(* IEC 61131-3 sources: AXOpen/src/components.ur.robotics/ctrl/src/AxoUrCb3/v_3_x_x (part 2) *)

            Inputs.Zone                                             := Inputs.Inputs.Ints.Register_0;
            Inputs.InPosition                                       := Inputs.Inputs.Ints.Register_1;

           //Movement parameters
            Inputs.ActionNo                                         := Inputs.Inputs.Ints.Register_2;
            Inputs.GlobalSpeed                                      := Inputs.Inputs.Ints.Register_3;
            Inputs.ToolNo                                           := Inputs.Inputs.Ints.Register_4;
            Inputs.WorkobjectNo                                     := Inputs.Inputs.Ints.Register_5;
            Inputs.PointNo                                          := Inputs.Inputs.Ints.Register_6;

            Inputs.UserSpecSpeed1                                   := Inputs.Inputs.Floats.Register_0;
            Inputs.UserSpecSpeed2                                   := Inputs.Inputs.Floats.Register_1;
            Inputs.Coordinates.X                                    := Inputs.Inputs.Floats.Register_2;
            Inputs.Coordinates.Y                                    := Inputs.Inputs.Floats.Register_3;
            Inputs.Coordinates.Z                                    := Inputs.Inputs.Floats.Register_4;
            Inputs.Coordinates.Rx                                   := Inputs.Inputs.Floats.Register_5;
            Inputs.Coordinates.Ry                                   := Inputs.Inputs.Floats.Register_6;
            Inputs.Coordinates.Rz                                   := Inputs.Inputs.Floats.Register_7;

            //*************StartAtMainTask***************
            StartAtMainTask.SetIsDisabled(_stopTasksAreActive);
            IF StartAtMainTask.StartTriggered() THEN
                Status.Action.Id :=  UINT#100;
            END_IF;
            Messenger.ActivateOnCondition(ULINT#100,StartAtMainTask.IsBusy(), eAxoMessageCategory#Info);
            Messenger.ActivateOnCondition(ULINT#101,StartAtMainTask.IsDone(), eAxoMessageCategory#Info);
            IF StartAtMainTask.Execute(THIS) THEN
                _blink.Blink(Context := _context, inOnTime:=T#500MS,inOffTime:=T#500MS);
                IF _power_progress = 0 THEN
                    Status.Error.Id := UINT#0;
                    TaskMessenger.Restore();
                    THIS.CallTimers(FALSE);
                    _power_progress := 300;
                END_IF;
                // Start at main running: waiting for 'NORMAL' or 'REDUCED' mode is choosen.
                IF _power_progress = 300 THEN
                    IF _infoTimer.output THEN
                        IF NOT Inputs.Inputs.Safety.NO_IsNormalMode THEN
                            TaskMessenger.Activate( UINT#500, eAxoMessageCategory#Potential);
                            Status.Error.Id :=      UINT#500;
                        END_IF;
                        IF NOT Inputs.Inputs.Safety.RD_IsReducedMode THEN
                            TaskMessenger.Activate( UINT#501, eAxoMessageCategory#Potential);
                            Status.Error.Id :=      UINT#501;
                        END_IF;
                    END_IF;

                    IF Inputs.Inputs.Safety.NO_IsNormalMode OR Inputs.Inputs.Safety.RD_IsReducedMode THEN
                        THIS.CallTimers(FALSE);
                        _power_progress:=302;
                    END_IF;
                END_IF;
                // Start at main running: waiting for the program to start running.
                IF _power_progress = 302 THEN
                    IF _infoTimer.output THEN
                        TaskMessenger.Activate( UINT#502, eAxoMessageCategory#Potential);
                        Status.Error.Id :=      UINT#502;
                    END_IF;

                    Outputs.Start:=_blink.output;

                    IF Inputs.Inputs.Robot.PR_IsProgramRunning THEN
                        Outputs.Start := FALSE;
                        THIS.CallTimers(FALSE);
                        _power_progress:=303;
                    END_IF;
                END_IF;
                // Start at main finished.
                IF _power_progress = 303 THEN
                    StartAtMainTask.DoneWhen(TRUE);
                    THIS.CallTimers(FALSE);
                    _power_progress := 0;
                END_IF;

                THIS.CallTimers(TRUE);
                StartAtMainTask.ThrowWhen(_errorTimer.output );
                Status.Action.Id := TO_UINT(_power_progress);
                StartAtMainTask.ThrowWhen(StartAtMainTask.Duration >= Config.TaskTimeout AND Config.TaskTimeout > T#0s ,'<#StartAtMainTask timeout.#>');
            END_IF;
            IF StartAtMainTask.DoneReached() THEN
                Status.Action.Id :=  UINT#101;
                Status.Error.Id :=  UINT#0;
            ELSIF StartAtMainTask.ErrorOccured() THEN
                Status.Action.Id :=  UINT#10000;
                Status.Error.Id  :=  UINT#10000;
            ELSIF StartAtMainTask.AbortTriggered()THEN
                Status.Action.Id :=  UINT#10001;
                Status.Error.Id  :=  UINT#10001;
            END_IF;
            Messenger.ActivateOnCondition(ULINT#10000,StartAtMainTask.HasError(), eAxoMessageCategory#Error);
            Messenger.ActivateOnCondition(ULINT#10001,StartAtMainTask.IsAborted(), eAxoMessageCategory#Info);
            Messenger.ActivateOnCondition(ULINT#102,StartAtMainTask.RestoreTriggered() , eAxoMessageCategory#Info);
            IF StartAtMainTask.RestoreTriggered() AND _power_progress >= 300 AND _power_progress <= 309  THEN
                Status.Action.Id :=  UINT#102;
                _power_progress := 0;
            END_IF;
            //*******************************************

            //***********StartMotorsAndProgramTask*******
            StartMotorsAndProgramTask.SetIsDisabled(_stopTasksAreActive);
            IF StartMotorsAndProgramTask.StartTriggered() THEN
                Status.Action.Id :=  UINT#110;
            END_IF;
            Messenger.ActivateOnCondition(ULINT#110,StartMotorsAndProgramTask.IsBusy(), eAxoMessageCategory#Info);
            Messenger.ActivateOnCondition(ULINT#111,StartMotorsAndProgramTask.IsDone(), eAxoMessageCategory#Info);
            IF StartMotorsAndProgramTask.Execute(THIS) THEN
                _blink.Blink(Context := _context, inOnTime:=T#500MS,inOffTime:=T#500MS);

                IF _power_progress = 0 THEN
                    Status.Error.Id := UINT#0;
                    TaskMessenger.Restore();
                    THIS.CallTimers(FALSE);
                    _power_progress := 310;
                END_IF;
                // Start motors and program running: waiting for 'NORMAL' or 'REDUCED' mode is choosen.
                IF _power_progress = 310 THEN
                    IF _infoTimer.output THEN
                        IF NOT Inputs.Inputs.Safety.NO_IsNormalMode THEN
                            TaskMessenger.Activate( UINT#510, eAxoMessageCategory#Potential);
                            Status.Error.Id :=      UINT#510;
                        END_IF;
                        IF NOT Inputs.Inputs.Safety.RD_IsReducedMode THEN
                            TaskMessenger.Activate( UINT#511, eAxoMessageCategory#Potential);
                            Status.Error.Id :=      UINT#511;
                        END_IF;
                    END_IF;

                    IF Inputs.Inputs.Safety.NO_IsNormalMode OR Inputs.Inputs.Safety.RD_IsReducedMode THEN
                        THIS.CallTimers(FALSE);
                        _power_progress:=312;
                    END_IF;
                END_IF;
                // Start motors and program running: waiting for the error to be reset (on the robot teach pendant).
                IF _power_progress = 312 THEN
                    IF _infoTimer.output THEN
                        TaskMessenger.Activate( UINT#512, eAxoMessageCategory#Potential);
                        Status.Error.Id :=      UINT#512;
                    END_IF;

                    IF NOT Inputs.Inputs.Safety.FT_IsFault THEN
                        THIS.CallTimers(FALSE);
                        _power_progress := 313;
                    END_IF;
                END_IF;
                // Start motors and program running: waiting for the emergency stop error to be reset (on the robot teach pendant).
                IF _power_progress = 313 THEN
                    IF _infoTimer.output THEN
                        IF Inputs.Inputs.Safety.ES_IsEmergencyStopped  THEN
                            TaskMessenger.Activate( UINT#513, eAxoMessageCategory#Potential);
                            Status.Error.Id :=      UINT#513;
                        END_IF;
                        IF Inputs.Inputs.Safety.PS_IsProtectiveStopped  THEN
                            TaskMessenger.Activate( UINT#514, eAxoMessageCategory#Potential);
                            Status.Error.Id :=      UINT#514;
                        END_IF;
                        IF Inputs.Inputs.Safety.SS_IsSafeguardStopped  THEN
                            TaskMessenger.Activate( UINT#515, eAxoMessageCategory#Potential);
                            Status.Error.Id :=      UINT#515;
                        END_IF;
                        IF Inputs.Inputs.Safety.RC_IsRecoveryMode  THEN
                            TaskMessenger.Activate( UINT#516, eAxoMessageCategory#Potential);
                            Status.Error.Id :=      UINT#516;
                        END_IF;
                        IF Inputs.Inputs.Safety.ST_IsStoppedDueSafety  THEN
                            TaskMessenger.Activate( UINT#517, eAxoMessageCategory#Potential);
                            Status.Error.Id :=      UINT#517;
                        END_IF;
                        IF Inputs.Inputs.Safety.VL_IsViolation  THEN
                            TaskMessenger.Activate( UINT#518, eAxoMessageCategory#Potential);
                            Status.Error.Id :=      UINT#518;
                        END_IF;
                    END_IF;

                    IF NOT Inputs.Inputs.Safety.ES_IsEmergencyStopped
                        AND NOT Inputs.Inputs.Safety.PS_IsProtectiveStopped
                        AND NOT Inputs.Inputs.Safety.SS_IsSafeguardStopped
                        AND NOT Inputs.Inputs.Safety.RC_IsRecoveryMode
                        AND NOT Inputs.Inputs.Safety.ST_IsStoppedDueSafety
                        AND NOT Inputs.Inputs.Safety.VL_IsViolation THEN
                        THIS.CallTimers(FALSE);
                        _power_progress := 319;
                    END_IF;
                END_IF;
                // Start motors and program running: waiting for the motors to be powered on.
                IF _power_progress = 319 THEN
                    IF _infoTimer.output THEN
                        TaskMessenger.Activate( UINT#519, eAxoMessageCategory#Potential);
                        Status.Error.Id :=      UINT#519;
                    END_IF;

                    Outputs.MotorOn:=_blink.output;

                    IF Inputs.Inputs.Safety.FT_IsFault THEN
                        THIS.CallTimers(FALSE);
                        _power_progress := 310;
                    END_IF;

                    IF Inputs.Inputs.Robot.PW_IsPowerOn THEN
                         Outputs.MotorOn:=FALSE;
                         THIS.CallTimers(FALSE);
                         _power_progress := 320;
                    END_IF;
                END_IF;
                // Start motors and program running: waiting for the motors to be powered on.
                IF _power_progress = 320 THEN
                    IF _infoTimer.output THEN
                        TaskMessenger.Activate( UINT#520, eAxoMessageCategory#Potential);
                        Status.Error.Id :=      UINT#520;
                    END_IF;

                    Outputs.MotorOn:=_blink.output;

                    IF Inputs.Inputs.Safety.FT_IsFault THEN
                        THIS.CallTimers(FALSE);
                        _power_progress := 310;
                    END_IF;

                    IF Inputs.Inputs.Robot.PW_IsPowerOn THEN
                         Outputs.MotorOn:=FALSE;
                         THIS.CallTimers(FALSE);
                         _power_progress := 321;
                    END_IF;
                END_IF;
                // Start motors and program running: waiting for the program to start running.
                IF _power_progress = 321 THEN
                    IF _infoTimer.output THEN
                        TaskMessenger.Activate( UINT#521, eAxoMessageCategory#Potential);
                        Status.Error.Id :=      UINT#521;
                    END_IF;

                    Outputs.Start:=_blink.output;

                    IF Inputs.Inputs.Safety.FT_IsFault THEN
                        THIS.CallTimers(FALSE);
                        _power_progress := 310;
                    END_IF;

                    IF Inputs.Inputs.Robot.PR_IsProgramRunning AND NOT Inputs.Inputs.Safety.FT_IsFault THEN
                         Outputs.Start:=FALSE;
                         THIS.CallTimers(FALSE);
                         _power_progress := 322;
                    END_IF;
                END_IF;
                // Start motors and program finished.
                IF _power_progress = 322 THEN
                    StartMotorsAndProgramTask.DoneWhen(TRUE);
                    THIS.CallTimers(FALSE);
                    _power_progress := 0;
                END_IF;

                THIS.CallTimers(TRUE);
                StartMotorsAndProgramTask.ThrowWhen(_errorTimer.output);
                Status.Action.Id := TO_UINT(_power_progress);
                StartMotorsAndProgramTask.ThrowWhen(StartMotorsAndProgramTask.Duration >= Config.TaskTimeout AND Config.TaskTimeout > T#0s ,'<#StartMotorsAndProgramTask timeout.#>');
            END_IF;
            IF StartMotorsAndProgramTask.DoneReached() THEN
                Status.Action.Id :=  UINT#111;
                Status.Error.Id :=  UINT#0;
            ELSIF StartMotorsAndProgramTask.ErrorOccured() THEN
                Status.Action.Id :=  UINT#10010;
                Status.Error.Id  :=  UINT#10010;
            ELSIF StartMotorsAndProgramTask.AbortTriggered() THEN
                Status.Action.Id :=  UINT#10011;
                Status.Error.Id  :=  UINT#10011;
            END_IF;
            Messenger.ActivateOnCondition(ULINT#10010,StartMotorsAndProgramTask.HasError(), eAxoMessageCategory#Error);
            Messenger.ActivateOnCondition(ULINT#10011,StartMotorsAndProgramTask.IsAborted(), eAxoMessageCategory#Info);
            Messenger.ActivateOnCondition(ULINT#112,StartMotorsAndProgramTask.RestoreTriggered() , eAxoMessageCategory#Info);
            IF StartMotorsAndProgramTask.RestoreTriggered() AND _power_progress >= 310 AND _power_progress <= 329  THEN
                Status.Action.Id :=  UINT#112;
                _power_progress := 0;
            END_IF;
            //*******************************************

            //***********StartMovementsTask**************
            StartMovementsTask.SetIsDisabled(NOT Inputs.Inputs.Robot.PW_IsPowerOn);
            IF StartMovementsTask.StartTriggered() THEN
                Status.Action.Id :=  UINT#180;
            END_IF;
            Messenger.ActivateOnCondition(ULINT#180,StartMovementsTask.IsBusy(), eAxoMessageCategory#Info);
            Messenger.ActivateOnCondition(ULINT#181,StartMovementsTask.IsDone(), eAxoMessageCategory#Info);
            IF StartMovementsTask.Execute(THIS) THEN
                IF _movement_progress = 0 THEN
                    Status.Error.Id :=  UINT#0;
                    TaskMessenger.Restore();
                    THIS.CallTimers(FALSE);
                    _movement_progress := 380;
                END_IF;
                // Start movements running: waiting for the program to start running.
                IF _movement_progress = 380 THEN
                    IF _infoTimer.output THEN
                        TaskMessenger.Activate( UINT#580, eAxoMessageCategory#Potential);
                        Status.Error.Id :=      UINT#580;
                    END_IF;

                    IF Inputs.Inputs.Robot.PR_IsProgramRunning THEN
                        THIS.CallTimers(FALSE);
                        _movement_progress := 381;
                    END_IF;
                END_IF;
                // Start movements running: waiting for the motors to be powered on.
                IF _movement_progress = 381 THEN
                    IF _infoTimer.output THEN
                        TaskMessenger.Activate( UINT#581, eAxoMessageCategory#Potential);
                        Status.Error.Id :=      UINT#581;
                    END_IF;

                    IF Inputs.Inputs.Robot.PW_IsPowerOn THEN
                        THIS.CallTimers(FALSE);
                        _movement_progress := 382;
                    END_IF;
                END_IF;
                // Start movements running: waiting for the error to be reset (on the robot teach pendant).
                IF _movement_progress = 382 THEN
                    IF _infoTimer.output THEN
                        TaskMessenger.Activate( UINT#582, eAxoMessageCategory#Potential);
                        Status.Error.Id :=      UINT#582;
                    END_IF;

                    IF NOT Inputs.Inputs.Safety.FT_IsFault THEN
                        THIS.CallTimers(FALSE);
                        _movement_progress := 383;
                    END_IF;
                END_IF;
                // Start movements running: sending parameters of the movement to the controller.
                IF _movement_progress = 383 THEN
                    IF _infoTimer.output THEN
                        TaskMessenger.Activate( UINT#583, eAxoMessageCategory#Potential);
                        Status.Error.Id :=      UINT#583;
                    END_IF;

                    Outputs.GlobalSpeed     := TO_DINT(Status.CurrentMovementParameters.GlobalSpeed);
                    Outputs.ToolNo          := TO_DINT(Status.CurrentMovementParameters.ToolNo);
                    Outputs.WorkobjectNo    := TO_DINT(Status.CurrentMovementParameters.WorkobjectNo);
                    Outputs.PointNo         := TO_DINT(Status.CurrentMovementParameters.PointNo);
                    Outputs.UserSpecSpeed1  := Status.CurrentMovementParameters.UserSpecSpeed1;
                    Outputs.UserSpecSpeed2  := Status.CurrentMovementParameters.UserSpecSpeed2;
                    Outputs.Coordinates     := Status.CurrentMovementParameters.Coordinates;

                    Outputs.ActionNo := DINT#254;

                    IF Outputs.ActionNo = Inputs.ActionNo THEN
                        THIS.CallTimers(FALSE);
                        _movement_progress := 384;
                    END_IF;
                END_IF;
                // Start movements running: waiting for the movement parameters sent to the controller to be mirrored back.
                IF _movement_progress = 384 THEN
                    IF _infoTimer.output THEN
                        IF Inputs.GlobalSpeed <> TO_DINT(Status.CurrentMovementParameters.GlobalSpeed) THEN
                            TaskMessenger.Activate( UINT#584, eAxoMessageCategory#Potential);
                            Status.Error.Id :=      UINT#584;//<#Waiting for Inputs.GlobalSpeed to be equal to MovementParameters.GlobalSpeed!
                        END_IF;
                        IF Inputs.ToolNo <> TO_DINT(Status.CurrentMovementParameters.ToolNo) THEN
                            TaskMessenger.Activate( UINT#585, eAxoMessageCategory#Potential);
                            Status.Error.Id :=      UINT#585;//<#Waiting for Inputs.ToolNo to be equal to MovementParameters.ToolNo!
                        END_IF;
                        IF Inputs.WorkobjectNo <> TO_DINT(Status.CurrentMovementParameters.WorkobjectNo) THEN
                            TaskMessenger.Activate( UINT#586, eAxoMessageCategory#Potential);
                            Status.Error.Id :=      UINT#586;//<#Waiting for Inputs.WorkobjectNo to be equal to MovementParameters.WorkobjectNo!
                        END_IF;
                        IF Inputs.PointNo <> TO_DINT(Status.CurrentMovementParameters.PointNo) THEN
                            TaskMessenger.Activate( UINT#587, eAxoMessageCategory#Potential);
                            Status.Error.Id :=      UINT#587;//<#Waiting for Inputs.PointNo to be equal to MovementParameters.PointNo!
                        END_IF;
                        IF Inputs.UserSpecSpeed1 <> Status.CurrentMovementParameters.UserSpecSpeed1 THEN
                            TaskMessenger.Activate( UINT#588, eAxoMessageCategory#Potential);
                            Status.Error.Id :=      UINT#588;//<#Waiting for Inputs.UserSpecSpeed1 to be equal to MovementParameters.UserSpecSpeed1!
                        END_IF;
                        IF Inputs.UserSpecSpeed2 <> Status.CurrentMovementParameters.UserSpecSpeed2 THEN
                            TaskMessenger.Activate( UINT#589, eAxoMessageCategory#Potential);
                            Status.Error.Id :=      UINT#589;//<#Waiting for Inputs.UserSpecSpeed2 to be equal to MovementParameters.UserSpecSpeed2!
                        END_IF;
                    END_IF;

                    IF 	Inputs.GlobalSpeed      = TO_DINT(Status.CurrentMovementParameters.GlobalSpeed) AND
                        Inputs.ToolNo           = TO_DINT(Status.CurrentMovementParameters.ToolNo) AND
                        Inputs.WorkobjectNo     = TO_DINT(Status.CurrentMovementParameters.WorkobjectNo) AND
                        Inputs.PointNo          = TO_DINT(Status.CurrentMovementParameters.PointNo) AND
                        Inputs.UserSpecSpeed1   = Status.CurrentMovementParameters.UserSpecSpeed1 AND
                        Inputs.UserSpecSpeed2   = Status.CurrentMovementParameters.UserSpecSpeed2 AND
                        AXOpen.Components.Robotics.CoordinatesAreNearlyEqual(Inputs.Coordinates,Status.CurrentMovementParameters.Coordinates,REAL#0.01,REAL#0.01,REAL#0.01,REAL#0.01,REAL#0.01,REAL#0.01) THEN
                        THIS.CallTimers(FALSE);
                        _movement_progress:=390;
                    END_IF;
                END_IF;
                // Start movements running: acknowleadging of the movement parameters.
                IF _movement_progress = 390 THEN
                    IF _infoTimer.output THEN
                        TaskMessenger.Activate( UINT#590, eAxoMessageCategory#Potential);
                        Status.Error.Id :=      UINT#590;
                    END_IF;

                    Outputs.ActionNo := DINT#255;

                    IF Outputs.ActionNo = Inputs.ActionNo THEN
                        THIS.CallTimers(FALSE);
                        _movement_progress:=391;
                    END_IF;
                END_IF;
                // Start movements running: waiting for the movement is finished.
                IF _movement_progress = 391 THEN
                    IF _infoTimer.output THEN
                        TaskMessenger.Activate( UINT#591, eAxoMessageCategory#Potential);
                        Status.Error.Id :=      UINT#591;
                    END_IF;

                    Outputs.ActionNo := TO_DINT(Status.CurrentMovementParameters.ActionNo);

                    IF Outputs.ActionNo = Inputs.ActionNo THEN
                        THIS.CallTimers(FALSE);
                        _movement_progress:=392;
                    END_IF;
                END_IF;
                // Start movements running: acknowleadging of the finished movement.
                IF _movement_progress = 392 THEN
                    IF _infoTimer.output THEN
                        TaskMessenger.Activate( UINT#592, eAxoMessageCategory#Potential);
                        Status.Error.Id :=      UINT#592;
                    END_IF;

                    Outputs.ActionNo := DINT#255;

                    IF Outputs.ActionNo = Inputs.ActionNo THEN
                        _movement_progress := 0;
                        StartMovementsTask.DoneWhen(TRUE);
                    END_IF;
                END_IF;

	            THIS.CallTimers(TRUE);

                StartMovementsTask.ThrowWhen(_errorTimer.output);
                Status.Action.Id := TO_UINT(_movement_progress);
                StartMovementsTask.ThrowWhen(StartMovementsTask.Duration >= Config.TaskTimeout AND Config.TaskTimeout > T#0s ,'<#StartMovementsTask timeout.#>');
            END_IF;
            IF StartMovementsTask.DoneReached() THEN
                Status.Action.Id :=  UINT#181;
                Status.Error.Id :=  UINT#0;
            ELSIF StartMovementsTask.ErrorOccured() THEN
                Status.Action.Id :=  UINT#10080;
                Status.Error.Id  :=  UINT#10080;
            ELSIF StartMovementsTask.AbortTriggered()THEN
                Status.Action.Id :=  UINT#10081;
                Status.Error.Id  :=  UINT#10081;
            END_IF;
            Messenger.ActivateOnCondition(ULINT#10080,StartMovementsTask.HasError(), eAxoMessageCategory#Error);
            Messenger.ActivateOnCondition(ULINT#10081,StartMovementsTask.IsAborted(), eAxoMessageCategory#Info);
            Messenger.ActivateOnCondition(ULINT#182,StartMovementsTask.RestoreTriggered() , eAxoMessageCategory#Info);
            IF StartMovementsTask.RestoreTriggered() AND _movement_progress >= 380 AND _movement_progress <= 399  THEN
                Status.Action.Id :=  UINT#182;
                _movement_progress := 0;
            END_IF;
            //*******************************************

            //***********StopMovementsAndProgramTask*****
            StopMovementsAndProgramTask.SetIsDisabled(FALSE);
            IF StopMovementsAndProgramTask.StartTriggered() THEN
                Status.Action.Id :=  UINT#210;
            END_IF;
            Messenger.ActivateOnCondition(ULINT#210,StopMovementsAndProgramTask.IsBusy(), eAxoMessageCategory#Info);
            Messenger.ActivateOnCondition(ULINT#211,StopMovementsAndProgramTask.IsDone(), eAxoMessageCategory#Info);
            IF StopMovementsAndProgramTask.Execute(THIS) THEN
                IF _power_progress = 0 THEN
                    Status.Error.Id :=  UINT#0;
                    TaskMessenger.Restore();
                    THIS.CallTimers(FALSE);
                    _power_progress := 410;
                END_IF;
                // Stop movements and program running: waiting for 'NORMAL' or 'REDUCED' mode is choosen.
                IF _power_progress = 410 THEN
                    IF _infoTimer.output THEN
                        IF NOT Inputs.Inputs.Safety.NO_IsNormalMode THEN
                            TaskMessenger.Activate( UINT#610, eAxoMessageCategory#Potential);
                            Status.Error.Id :=      UINT#610;
                        END_IF;
                        IF NOT Inputs.Inputs.Safety.RD_IsReducedMode THEN
                            TaskMessenger.Activate( UINT#611, eAxoMessageCategory#Potential);
                            Status.Error.Id :=      UINT#611;
                        END_IF;
                    END_IF;

                    IF Inputs.Inputs.Safety.NO_IsNormalMode OR Inputs.Inputs.Safety.RD_IsReducedMode THEN
                        THIS.CallTimers(FALSE);
                        _power_progress:=412;
                    END_IF;
                END_IF;
                // Stop movements and program running: waiting for the program to be stopped."
                IF _power_progress = 412 THEN
                    IF _infoTimer.output THEN
                        TaskMessenger.Activate( UINT#612, eAxoMessageCategory#Potential);
                        Status.Error.Id :=      UINT#612;
                    END_IF;

                    Outputs.Stop := TRUE;

                    IF NOT Inputs.Inputs.Robot.PR_IsProgramRunning THEN
                        Outputs.Stop := FALSE ;
                        THIS.CallTimers(FALSE);
                        _power_progress:=413;
                    END_IF;
                END_IF;
                // Stop movements and program finished.
                IF _power_progress = 413 THEN
                    Outputs.Stop := FALSE ;
                    StopMovementsAndProgramTask.DoneWhen(TRUE);
                    _power_progress := 0;
                END_IF;

                THIS.CallTimers(TRUE);
                StopMovementsAndProgramTask.ThrowWhen(_errorTimer.output);
                Status.Action.Id := TO_UINT(_power_progress);
                StopMovementsAndProgramTask.ThrowWhen(StopMovementsAndProgramTask.Duration >= Config.TaskTimeout AND Config.TaskTimeout > T#0s ,'<#StopMovementsAndProgramTask timeout.#>');
            END_IF;
            IF StopMovementsAndProgramTask.DoneReached() THEN
                Status.Action.Id :=  UINT#211;
                Status.Error.Id :=  UINT#0;
            ELSIF StopMovementsAndProgramTask.ErrorOccured() THEN
                Status.Action.Id :=  UINT#10110;
                Status.Error.Id  :=  UINT#10110;
            ELSIF StopMovementsAndProgramTask.AbortTriggered()THEN
                Status.Action.Id :=  UINT#10111;
                Status.Error.Id  :=  UINT#10111;
            END_IF;
            Messenger.ActivateOnCondition(ULINT#10110,StopMovementsAndProgramTask.HasError(), eAxoMessageCategory#Error);
            Messenger.ActivateOnCondition(ULINT#10111,StopMovementsAndProgramTask.IsAborted(), eAxoMessageCategory#Info);
            Messenger.ActivateOnCondition(ULINT#212,StopMovementsAndProgramTask.RestoreTriggered() , eAxoMessageCategory#Info);
            IF StopMovementsAndProgramTask.RestoreTriggered() AND _power_progress >= 410 AND _power_progress <= 419  THEN
                Status.Action.Id :=  UINT#212;
                _power_progress := 0;
            END_IF;
            //*******************************************

            //***********StopMovementsTask***************
            StopMovementsTask.SetIsDisabled(FALSE);
            IF StopMovementsAndProgramTask.StartTriggered() THEN
                Status.Action.Id :=  UINT#220;
            END_IF;
            Messenger.ActivateOnCondition(ULINT#220,StopMovementsAndProgramTask.IsBusy(), eAxoMessageCategory#Info);
            Messenger.ActivateOnCondition(ULINT#221,StopMovementsAndProgramTask.IsDone(), eAxoMessageCategory#Info);
            IF StopMovementsTask.Execute(THIS) THEN
                IF _power_progress = 0 THEN
                    Status.Error.Id :=  UINT#0;
                    TaskMessenger.Restore();
                    THIS.CallTimers(FALSE);
                    _power_progress := 420;
                END_IF;
                // Stop movements running: waiting for 'NORMAL' or 'REDUCED' mode is choosen.
                IF _power_progress = 420 THEN
                    IF _infoTimer.output THEN
                        IF NOT Inputs.Inputs.Safety.NO_IsNormalMode THEN
                            TaskMessenger.Activate( UINT#620, eAxoMessageCategory#Potential);
                            Status.Error.Id :=      UINT#620;
                        END_IF;
                        IF NOT Inputs.Inputs.Safety.RD_IsReducedMode THEN
                            TaskMessenger.Activate( UINT#621, eAxoMessageCategory#Potential);
                            Status.Error.Id :=      UINT#621;
                        END_IF;
                    END_IF;

                    IF Inputs.Inputs.Safety.NO_IsNormalMode OR Inputs.Inputs.Safety.RD_IsReducedMode THEN
                        THIS.CallTimers(FALSE);
                        _power_progress:=422;
                    END_IF;
                END_IF;
                // Stop movements running: waiting for the program to be stopped.
                IF _power_progress = 422 THEN
                    IF _infoTimer.output THEN
                        TaskMessenger.Activate( UINT#622, eAxoMessageCategory#Potential);
                        Status.Error.Id :=      UINT#622;
                    END_IF;

                    Outputs.Pause := TRUE;

                    IF NOT Inputs.Inputs.Robot.PR_IsProgramRunning THEN
                        Outputs.Pause := FALSE ;
                        THIS.CallTimers(FALSE);
                        _power_progress:=423;
                    END_IF;
                END_IF;
                // Stop movements finished.
                IF _power_progress = 423 THEN
                    Outputs.Pause := FALSE ;
                    StopMovementsTask.DoneWhen(TRUE);
                    _power_progress := 0;
                END_IF;

                THIS.CallTimers(TRUE);
                StopMovementsTask.ThrowWhen(_errorTimer.output);
                Status.Action.Id := TO_UINT(_power_progress);
                StopMovementsTask.ThrowWhen(StopMovementsTask.Duration >= Config.TaskTimeout AND Config.TaskTimeout > T#0s ,'<#StopMovementsTask timeout.#>');
            END_IF;
            IF StopMovementsTask.DoneReached() THEN
                Status.Action.Id :=  UINT#221;
                Status.Error.Id :=  UINT#0;
            ELSIF StopMovementsTask.ErrorOccured() THEN
                Status.Action.Id :=  UINT#10120;
                Status.Error.Id  :=  UINT#10120;
            ELSIF StopMovementsTask.AbortTriggered()THEN
                Status.Action.Id :=  UINT#10121;
                Status.Error.Id  :=  UINT#10121;
            END_IF;
            Messenger.ActivateOnCondition(ULINT#10120,StopMovementsTask.HasError(), eAxoMessageCategory#Error);
            Messenger.ActivateOnCondition(ULINT#10121,StopMovementsTask.IsAborted(), eAxoMessageCategory#Info);
            Messenger.ActivateOnCondition(ULINT#222,StopMovementsTask.RestoreTriggered() , eAxoMessageCategory#Info);
            IF StopMovementsTask.RestoreTriggered() AND _power_progress >= 420 AND _power_progress <= 429  THEN
                Status.Action.Id :=  UINT#222;
                _power_progress := 0;
            END_IF;
            //*******************************************

            //*************POWER ON********************
            PowerOnTask.SetIsDisabled(NOT(Inputs.RobotMode=eAxoUrRoboticsRobotMode#DISCONNECTED AND Config.RemotePowerOnEnabled));
            IF PowerOnTask.Execute(THIS) THEN
                refPowerOnPulse^ :=TRUE;
                Status.Action.Id :=  UINT#420;//('<#POWER ON PULSE WAS SEND TO CONTROLER#>');
                PowerOnTask.DoneWhen(PowerOnTask.Duration > Config.RemotePowerOnPulse);
            END_IF;

            IF refPowerOnPulse^ AND PowerOnTask.IsDone()  OR NOT Config.RemotePowerOnEnabled THEN
                refPowerOnPulse^ :=FALSE;
            END_IF;

            //****************************************

            _someTaskIsActive := StartAtMainTask.IsBusy()
                                OR StartMotorsAndProgramTask.IsBusy()
                                OR StartMovementsTask.IsBusy()
                                OR StopMovementsTask.IsBusy()
                                OR StopMovementsAndProgramTask.IsBusy();

            IF _someTaskIsActive THEN
                IF(Inputs.Inputs.Safety.ES_IsEmergencyStopped) THEN
                    Messenger.Activate(UINT#2000, eAxoMessageCategory#Error);
                    Status.Error.Id := UINT#2000;
                END_IF;
                IF(Inputs.Inputs.Safety.ST_IsStoppedDueSafety) THEN
                    Messenger.Activate(UINT#2001, eAxoMessageCategory#Error);
                    Status.Error.Id := UINT#2001;
                END_IF;
            END_IF;
            //***********UPDATE**OUTPUTS*****************
            //SYSTEM OUTPUTS
            Outputs.Outputs.Reg1.Bit_0 := Outputs.Start;
            Outputs.outputs.Reg1.Bit_1 := Outputs.Stop;
            Outputs.outputs.Reg1.Bit_2 := Outputs.Pause;
            Outputs.outputs.Reg1.Bit_3 := Outputs.MotorOn;
            //Outputs.outputs.Reg1.Bit_4 := Outputs.RunAction;

            //Tool signals
            Outputs.Outputs.Reg1.Bit_8 := Outputs.Tool_1_Retract;
            Outputs.outputs.Reg1.Bit_9 := Outputs.Tool_1_Extend;
            Outputs.outputs.Reg1.Bit_10 := Outputs.Tool_2_Retract;
            Outputs.outputs.Reg1.Bit_11 := Outputs.Tool_2_Extend;
            Outputs.outputs.Reg1.Bit_12 := Outputs.Tool_3_Retract;
            Outputs.outputs.Reg1.Bit_13 := Outputs.Tool_3_Extend;
            Outputs.outputs.Reg1.Bit_14 := Outputs.Tool_4_Retract;
            Outputs.outputs.Reg1.Bit_15 := Outputs.Tool_4_Extend;

            //zone
            Outputs.Outputs.Reg1.Int_0 := Outputs.Zone;
            //position
            Outputs.Outputs.Reg1.Int_1 := Outputs.InPosition;

            //Movement parameters
            Outputs.Outputs.Reg1.Int_2 := Outputs.ActionNo;
            Outputs.Outputs.Reg1.Int_3 := Outputs.GlobalSpeed;
            Outputs.Outputs.Reg1.Int_4 := Outputs.ToolNo;
            Outputs.Outputs.Reg1.Int_5 := Outputs.WorkobjectNo;
            Outputs.Outputs.Reg1.Int_6 := Outputs.PointNo;
            //master mode  such as manual/auto ....
            Outputs.Outputs.Reg1.Int_7 := TO_DINT(Outputs.MasterMode);

            Outputs.Outputs.Reg1.Float_0 := Outputs.UserSpecSpeed1;
            Outputs.Outputs.Reg1.Float_1 := Outputs.UserSpecSpeed2;

            ////Coordinates
            Outputs.Outputs.Reg1.Float_2 := Outputs.Coordinates.X ;
            Outputs.Outputs.Reg1.Float_3 := Outputs.Coordinates.Y;
            Outputs.Outputs.Reg1.Float_4 := Outputs.Coordinates.Z ;
            Outputs.Outputs.Reg1.Float_5 := (Outputs.Coordinates.Rx);
            Outputs.Outputs.Reg1.Float_6 := (Outputs.Coordinates.Ry);
            Outputs.Outputs.Reg1.Float_7 := (Outputs.Coordinates.Rz);

            //st_URO_CB3_O2TSpeedData => 8_O2T Robot IO
            _data24[0].%X0 := Outputs.Outputs.Speed.SSM_SpeedSliderFractionMask;

            _dword := TO_DWORD(Outputs.Outputs.Speed.SpeedSliderFraction * REAL#0.01);
            _data24[4] := _dword.%B3;
            _data24[5] := _dword.%B2;
            _data24[6] := _dword.%B1;
            _data24[7] := _dword.%B0;

            //st_URO_CB3_O2TIoData => 8_O2T Robot IO
            _data24[8]  := TO_BYTE(Outputs.Outputs.IO.StandardDigitalOutputMask);
            _data24[9]  := TO_BYTE(Outputs.Outputs.IO.ConfigurableDigitalOutputMask);
            _data24[10] := TO_BYTE(Outputs.Outputs.IO.StandardDigitalOutputs);
            _data24[11] := TO_BYTE(Outputs.Outputs.IO.ConfigurableDdigitalOutputs);
            _data24[12] := TO_BYTE(Outputs.Outputs.IO.AOM_AnalogOutputMask);
            _data24[13] := TO_BYTE(Outputs.Outputs.IO.AOT_AnalogOutputTypes);
            _data24[14] := TO_BYTE(Outputs.Outputs.IO.TDOM_ToolDigitalOutputMask);
            _data24[15] := TO_BYTE(Outputs.Outputs.IO.TDO_ToolDigitalOutput);

            _dword := TO_DWORD(Outputs.Outputs.IO.StandardAnalogOutput_0);
            _data24[16] := _dword.%B3;
            _data24[17] := _dword.%B2;
            _data24[18] := _dword.%B1;
            _data24[19] := _dword.%B0;

            _dword := TO_DWORD(Outputs.Outputs.IO.StandardAnalogOutput_1);
            _data24[20] := _dword.%B3;
            _data24[21] := _dword.%B2;
            _data24[22] := _dword.%B1;
            _data24[23] := _dword.%B0;

            _retVal := Siemens.Simatic.DistributedIO.WriteData((Config.HWIDs.HwId_AxoUrRobotics_O2T_Robot_IO),_data24);
            IF _retVal > WORD#0 THEN
                Messenger.Activate(UINT#1231, eAxoMessageCategory#Error);
                Status.Error.Id := UINT#1231;
                RETURN;
            END_IF;

            //st_URO_CB3_O2TRegData => 9_O2T General Purpose Registers 1
            _data100[0].%X0 :=  Outputs.Outputs.Reg1.Bit_0;
            _data100[0].%X1 :=  Outputs.Outputs.Reg1.Bit_1;
            _data100[0].%X2 :=  Outputs.Outputs.Reg1.Bit_2;
            _data100[0].%X3 :=  Outputs.Outputs.Reg1.Bit_3;
            _data100[0].%X4 :=  Outputs.Outputs.Reg1.Bit_4;
            _data100[0].%X5 :=  Outputs.Outputs.Reg1.Bit_5;
            _data100[0].%X6 :=  Outputs.Outputs.Reg1.Bit_6;
            _data100[0].%X7 :=  Outputs.Outputs.Reg1.Bit_7;

            _data100[1].%X0 :=  Outputs.Outputs.Reg1.Bit_8;
            _data100[1].%X1 :=  Outputs.Outputs.Reg1.Bit_9;
            _data100[1].%X2 :=  Outputs.Outputs.Reg1.Bit_10;
            _data100[1].%X3 :=  Outputs.Outputs.Reg1.Bit_11;
            _data100[1].%X4 :=  Outputs.Outputs.Reg1.Bit_12;
            _data100[1].%X5 :=  Outputs.Outputs.Reg1.Bit_13;
            _data100[1].%X6 :=  Outputs.Outputs.Reg1.Bit_14;
            _data100[1].%X7 :=  Outputs.Outputs.Reg1.Bit_15;

            _data100[2].%X0 :=  Outputs.Outputs.Reg1.Bit_16;
            _data100[2].%X1 :=  Outputs.Outputs.Reg1.Bit_17;
            _data100[2].%X2 :=  Outputs.Outputs.Reg1.Bit_18;
            _data100[2].%X3 :=  Outputs.Outputs.Reg1.Bit_19;
            _data100[2].%X4 :=  Outputs.Outputs.Reg1.Bit_20;
            _data100[2].%X5 :=  Outputs.Outputs.Reg1.Bit_21;
            _data100[2].%X6 :=  Outputs.Outputs.Reg1.Bit_22;
            _data100[2].%X7 :=  Outputs.Outputs.Reg1.Bit_23;

            _data100[3].%X0 :=  Outputs.Outputs.Reg1.Bit_24;
            _data100[3].%X1 :=  Outputs.Outputs.Reg1.Bit_25;
            _data100[3].%X2 :=  Outputs.Outputs.Reg1.Bit_26;
            _data100[3].%X3 :=  Outputs.Outputs.Reg1.Bit_27;
            _data100[3].%X4 :=  Outputs.Outputs.Reg1.Bit_28;
            _data100[3].%X5 :=  Outputs.Outputs.Reg1.Bit_29;
            _data100[3].%X6 :=  Outputs.Outputs.Reg1.Bit_30;
            _data100[3].%X7 :=  Outputs.Outputs.Reg1.Bit_31;

            _dword          := TO_DWORD( Outputs.Outputs.Reg1.Int_0);
            _data100[4]     := _dword.%B3;
            _data100[5]     := _dword.%B2;
            _data100[6]     := _dword.%B1;
            _data100[7]     := _dword.%B0;

            _dword          := TO_DWORD( Outputs.Outputs.Reg1.Int_1);
            _data100[8]     := _dword.%B3;
            _data100[9]     := _dword.%B2;
            _data100[10]    := _dword.%B1;
            _data100[11]    := _dword.%B0;

            _dword          := TO_DWORD( Outputs.Outputs.Reg1.Int_2);
            _data100[12]    := _dword.%B3;
            _data100[13]    := _dword.%B2;
            _data100[14]    := _dword.%B1;
            _data100[15]    := _dword.%B0;

            _dword          := TO_DWORD( Outputs.Outputs.Reg1.Int_3);
            _data100[16]    := _dword.%B3;
            _data100[17]    := _dword.%B2;
            _data100[18]    := _dword.%B1;
            _data100[19]    := _dword.%B0;

            _dword          := TO_DWORD( Outputs.Outputs.Reg1.Int_4);
            _data100[20]    := _dword.%B3;
            _data100[21]    := _dword.%B2;
            _data100[22]    := _dword.%B1;
            _data100[23]    := _dword.%B0;

            _dword          := TO_DWORD( Outputs.Outputs.Reg1.Int_5);
            _data100[24]    := _dword.%B3;
            _data100[25]    := _dword.%B2;
            _data100[26]    := _dword.%B1;
            _data100[27]    := _dword.%B0;

            _dword          := TO_DWORD( Outputs.Outputs.Reg1.Int_6);
            _data100[28]    := _dword.%B3;
            _data100[29]    := _dword.%B2;
            _data100[30]    := _dword.%B1;
            _data100[31]    := _dword.%B0;

            _dword          := TO_DWORD( Outputs.Outputs.Reg1.Int_7);
            _data100[32]    := _dword.%B3;
            _data100[33]    := _dword.%B2;
            _data100[34]    := _dword.%B1;
            _data100[35]    := _dword.%B0;

            _dword          := TO_DWORD( Outputs.Outputs.Reg1.Int_8);
            _data100[36]    := _dword.%B3;
            _data100[37]    := _dword.%B2;
            _data100[38]    := _dword.%B1;
            _data100[39]    := _dword.%B0;

            _dword          := TO_DWORD( Outputs.Outputs.Reg1.Int_9);
            _data100[40]    := _dword.%B3;
            _data100[41]    := _dword.%B2;
            _data100[42]    := _dword.%B1;
            _data100[43]    := _dword.%B0;

            _dword          := TO_DWORD( Outputs.Outputs.Reg1.Int_10);
            _data100[44]    := _dword.%B3;
            _data100[45]    := _dword.%B2;
            _data100[46]    := _dword.%B1;
            _data100[47]    := _dword.%B0;

            _dword          := TO_DWORD( Outputs.Outputs.Reg1.Int_11);
            _data100[48]    := _dword.%B3;
            _data100[49]    := _dword.%B2;
            _data100[50]    := _dword.%B1;
            _data100[51]    := _dword.%B0;

            _dword          := TO_DWORD( Outputs.Outputs.Reg1.Float_0);
            _data100[52]    := _dword.%B3;
            _data100[53]    := _dword.%B2;
            _data100[54]    := _dword.%B1;
            _data100[55]    := _dword.%B0;

            _dword          := TO_DWORD( Outputs.Outputs.Reg1.Float_1);
            _data100[56]    := _dword.%B3;
            _data100[57]    := _dword.%B2;
            _data100[58]    := _dword.%B1;
            _data100[59]    := _dword.%B0;

            _dword          := TO_DWORD( Outputs.Outputs.Reg1.Float_2);
            _data100[60]    := _dword.%B3;
            _data100[61]    := _dword.%B2;
            _data100[62]    := _dword.%B1;
            _data100[63]    := _dword.%B0;

            _dword          := TO_DWORD( Outputs.Outputs.Reg1.Float_3);
            _data100[64]    := _dword.%B3;
            _data100[65]    := _dword.%B2;
            _data100[66]    := _dword.%B1;
            _data100[67]    := _dword.%B0;

            _dword          := TO_DWORD( Outputs.Outputs.Reg1.Float_4);
            _data100[68]    := _dword.%B3;
            _data100[69]    := _dword.%B2;
            _data100[70]    := _dword.%B1;
            _data100[71]    := _dword.%B0;

            _dword          := TO_DWORD( Outputs.Outputs.Reg1.Float_5);
            _data100[72]    := _dword.%B3;
            _data100[73]    := _dword.%B2;
            _data100[74]    := _dword.%B1;
            _data100[75]    := _dword.%B0;

            _dword          := TO_DWORD( Outputs.Outputs.Reg1.Float_6);
            _data100[76]    := _dword.%B3;
            _data100[77]    := _dword.%B2;
            _data100[78]    := _dword.%B1;
            _data100[79]    := _dword.%B0;

            _dword          := TO_DWORD( Outputs.Outputs.Reg1.Float_7);
            _data100[80]    := _dword.%B3;
            _data100[81]    := _dword.%B2;
            _data100[82]    := _dword.%B1;
            _data100[83]    := _dword.%B0;

            _dword          := TO_DWORD( Outputs.Outputs.Reg1.Float_8);
            _data100[84]    := _dword.%B3;
            _data100[85]    := _dword.%B2;
            _data100[86]    := _dword.%B1;
            _data100[87]    := _dword.%B0;

            _dword          := TO_DWORD( Outputs.Outputs.Reg1.Float_9);
            _data100[88]    := _dword.%B3;
            _data100[89]    := _dword.%B2;
            _data100[90]    := _dword.%B1;
            _data100[91]    := _dword.%B0;

            _dword          := TO_DWORD( Outputs.Outputs.Reg1.Float_10);
            _data100[92]    := _dword.%B3;
            _data100[93]    := _dword.%B2;
            _data100[94]    := _dword.%B1;
            _data100[95]    := _dword.%B0;

            _dword          := TO_DWORD( Outputs.Outputs.Reg1.Float_11);
            _data100[96]    := _dword.%B3;
            _data100[97]    := _dword.%B2;
            _data100[98]    := _dword.%B1;
            _data100[99]    := _dword.%B0;

            _retVal := Siemens.Simatic.DistributedIO.WriteData((Config.HWIDs.HwId_AxoUrRobotics_O2T_General_Purpose_Registers_1),_data100);
            IF _retVal > WORD#0 THEN
                Messenger.Activate(UINT#1232, eAxoMessageCategory#Error);
                Status.Error.Id := UINT#1232;
                RETURN;
            END_IF;

            //st_URO_CB3_O2TRegData => 10_O2T General Purpose Registers 2
            _data100[0].%X0 :=  Outputs.Outputs.Reg2.Bit_0;
            _data100[0].%X1 :=  Outputs.Outputs.Reg2.Bit_1;
            _data100[0].%X2 :=  Outputs.Outputs.Reg2.Bit_2;
            _data100[0].%X3 :=  Outputs.Outputs.Reg2.Bit_3;
            _data100[0].%X4 :=  Outputs.Outputs.Reg2.Bit_4;
            _data100[0].%X5 :=  Outputs.Outputs.Reg2.Bit_5;
            _data100[0].%X6 :=  Outputs.Outputs.Reg2.Bit_6;
            _data100[0].%X7 :=  Outputs.Outputs.Reg2.Bit_7;

            _data100[1].%X0 :=  Outputs.Outputs.Reg2.Bit_8;
            _data100[1].%X1 :=  Outputs.Outputs.Reg2.Bit_9;
            _data100[1].%X2 :=  Outputs.Outputs.Reg2.Bit_10;
            _data100[1].%X3 :=  Outputs.Outputs.Reg2.Bit_11;
            _data100[1].%X4 :=  Outputs.Outputs.Reg2.Bit_12;
            _data100[1].%X5 :=  Outputs.Outputs.Reg2.Bit_13;
            _data100[1].%X6 :=  Outputs.Outputs.Reg2.Bit_14;
            _data100[1].%X7 :=  Outputs.Outputs.Reg2.Bit_15;

            _data100[2].%X0 :=  Outputs.Outputs.Reg2.Bit_16;
            _data100[2].%X1 :=  Outputs.Outputs.Reg2.Bit_17;
            _data100[2].%X2 :=  Outputs.Outputs.Reg2.Bit_18;
            _data100[2].%X3 :=  Outputs.Outputs.Reg2.Bit_19;
            _data100[2].%X4 :=  Outputs.Outputs.Reg2.Bit_20;
            _data100[2].%X5 :=  Outputs.Outputs.Reg2.Bit_21;
            _data100[2].%X6 :=  Outputs.Outputs.Reg2.Bit_22;
            _data100[2].%X7 :=  Outputs.Outputs.Reg2.Bit_23;

            _data100[3].%X0 :=  Outputs.Outputs.Reg2.Bit_24;
            _data100[3].%X1 :=  Outputs.Outputs.Reg2.Bit_25;
            _data100[3].%X2 :=  Outputs.Outputs.Reg2.Bit_26;
            _data100[3].%X3 :=  Outputs.Outputs.Reg2.Bit_27;
            _data100[3].%X4 :=  Outputs.Outputs.Reg2.Bit_28;
            _data100[3].%X5 :=  Outputs.Outputs.Reg2.Bit_29;
            _data100[3].%X6 :=  Outputs.Outputs.Reg2.Bit_30;
            _data100[3].%X7 :=  Outputs.Outputs.Reg2.Bit_31;

            _dword          := TO_DWORD( Outputs.Outputs.Reg2.Int_0);
            _data100[4]     := _dword.%B3;
            _data100[5]     := _dword.%B2;
            _data100[6]     := _dword.%B1;
            _data100[7]     := _dword.%B0;

            _dword          := TO_DWORD( Outputs.Outputs.Reg2.Int_1);
            _data100[8]     := _dword.%B3;
            _data100[9]     := _dword.%B2;
            _data100[10]    := _dword.%B1;
            _data100[11]    := _dword.%B0;

            _dword          := TO_DWORD( Outputs.Outputs.Reg2.Int_2);
            _data100[12]    := _dword.%B3;
            _data100[13]    := _dword.%B2;
            _data100[14]    := _dword.%B1;
            _data100[15]    := _dword.%B0;

            _dword          := TO_DWORD( Outputs.Outputs.Reg2.Int_3);
            _data100[16]    := _dword.%B3;
            _data100[17]    := _dword.%B2;
            _data100[18]    := _dword.%B1;
            _data100[19]    := _dword.%B0;

            _dword          := TO_DWORD( Outputs.Outputs.Reg2.Int_4);
            _data100[20]    := _dword.%B3;
            _data100[21]    := _dword.%B2;
            _data100[22]    := _dword.%B1;
            _data100[23]    := _dword.%B0;

            _dword          := TO_DWORD( Outputs.Outputs.Reg2.Int_5);
            _data100[24]    := _dword.%B3;
            _data100[25]    := _dword.%B2;
            _data100[26]    := _dword.%B1;
            _data100[27]    := _dword.%B0;

            _dword          := TO_DWORD( Outputs.Outputs.Reg2.Int_6);
            _data100[28]    := _dword.%B3;
            _data100[29]    := _dword.%B2;
            _data100[30]    := _dword.%B1;
            _data100[31]    := _dword.%B0;

            _dword          := TO_DWORD( Outputs.Outputs.Reg2.Int_7);
            _data100[32]    := _dword.%B3;
            _data100[33]    := _dword.%B2;
            _data100[34]    := _dword.%B1;
            _data100[35]    := _dword.%B0;

            _dword          := TO_DWORD( Outputs.Outputs.Reg2.Int_8);
            _data100[36]    := _dword.%B3;
            _data100[37]    := _dword.%B2;
            _data100[38]    := _dword.%B1;
            _data100[39]    := _dword.%B0;

            _dword          := TO_DWORD( Outputs.Outputs.Reg2.Int_9);
            _data100[40]    := _dword.%B3;
            _data100[41]    := _dword.%B2;
            _data100[42]    := _dword.%B1;
            _data100[43]    := _dword.%B0;

            _dword          := TO_DWORD( Outputs.Outputs.Reg2.Int_10);
            _data100[44]    := _dword.%B3;
            _data100[45]    := _dword.%B2;
            _data100[46]    := _dword.%B1;
            _data100[47]    := _dword.%B0;

            _dword          := TO_DWORD( Outputs.Outputs.Reg2.Int_11);
            _data100[48]    := _dword.%B3;
            _data100[49]    := _dword.%B2;
            _data100[50]    := _dword.%B1;
            _data100[51]    := _dword.%B0;

            _dword          := TO_DWORD( Outputs.Outputs.Reg2.Float_0);
            _data100[52]    := _dword.%B3;
            _data100[53]    := _dword.%B2;
            _data100[54]    := _dword.%B1;
            _data100[55]    := _dword.%B0;

            _dword          := TO_DWORD( Outputs.Outputs.Reg2.Float_1);
            _data100[56]    := _dword.%B3;
            _data100[58]    := _dword.%B2;
            _data100[58]    := _dword.%B1;
            _data100[59]    := _dword.%B0;

            _dword          := TO_DWORD( Outputs.Outputs.Reg2.Float_2);
            _data100[60]    := _dword.%B3;
            _data100[61]    := _dword.%B2;
            _data100[62]    := _dword.%B1;
            _data100[63]    := _dword.%B0;

            _dword          := TO_DWORD( Outputs.Outputs.Reg2.Float_3);
            _data100[64]    := _dword.%B3;
            _data100[65]    := _dword.%B2;
            _data100[66]    := _dword.%B1;
            _data100[67]    := _dword.%B0;

            _dword          := TO_DWORD( Outputs.Outputs.Reg2.Float_4);
            _data100[68]    := _dword.%B3;
            _data100[69]    := _dword.%B2;
            _data100[70]    := _dword.%B1;
            _data100[71]    := _dword.%B0;

            _dword          := TO_DWORD( Outputs.Outputs.Reg2.Float_5);
            _data100[72]    := _dword.%B3;
            _data100[73]    := _dword.%B2;
            _data100[74]    := _dword.%B1;
            _data100[75]    := _dword.%B0;

            _dword          := TO_DWORD( Outputs.Outputs.Reg2.Float_6);
            _data100[76]    := _dword.%B3;
            _data100[77]    := _dword.%B2;
            _data100[78]    := _dword.%B1;
            _data100[79]    := _dword.%B0;

            _dword          := TO_DWORD( Outputs.Outputs.Reg2.Float_7);
            _data100[80]    := _dword.%B3;
            _data100[81]    := _dword.%B2;
            _data100[82]    := _dword.%B1;
            _data100[83]    := _dword.%B0;

            _dword          := TO_DWORD( Outputs.Outputs.Reg2.Float_8);
            _data100[84]    := _dword.%B3;
            _data100[85]    := _dword.%B2;
            _data100[86]    := _dword.%B1;
            _data100[87]    := _dword.%B0;

            _dword          := TO_DWORD( Outputs.Outputs.Reg2.Float_9);
            _data100[88]    := _dword.%B3;
            _data100[89]    := _dword.%B2;
            _data100[90]    := _dword.%B1;
            _data100[91]    := _dword.%B0;

            _dword          := TO_DWORD( Outputs.Outputs.Reg2.Float_10);
            _data100[92]    := _dword.%B3;
            _data100[93]    := _dword.%B2;
            _data100[94]    := _dword.%B1;
            _data100[95]    := _dword.%B0;

            _dword          := TO_DWORD( Outputs.Outputs.Reg2.Float_11);
            _data100[96]    := _dword.%B3;
            _data100[97]    := _dword.%B2;
            _data100[98]    := _dword.%B1;
            _data100[99]    := _dword.%B0;

            _retVal := Siemens.Simatic.DistributedIO.WriteData((Config.HWIDs.HwId_AxoUrRobotics_O2T_General_Purpose_Registers_2),_data100);
            IF _retVal > WORD#0 THEN
                Messenger.Activate(UINT#1233, eAxoMessageCategory#Error);
                Status.Error.Id := UINT#1233;
                RETURN;
            END_IF;

        END_METHOD

        METHOD PROTECTED OVERRIDE ManualControl
            Status.CurrentMovementParameters := MovementParameters;
        END_METHOD

        ///<summary>
        /// Restores this component into intial state.
        ///</summary>
        METHOD PUBLIC OVERRIDE Restore
            PowerOnTask.Restore();
            StartAtMainTask.Restore();
            StartMotorsAndProgramTask.Restore();
            StopMovementsTask.Restore();
            StopMovementsAndProgramTask.Restore();
            StartMovementsTask.Restore();
	        RebootControllerTask.Restore();
            RestoreTask.DoneWhen(TRUE);
            Outputs.ActionNo:=255;
            Outputs.GlobalSpeed:=0;
            Outputs.ToolNo:=0;
            Outputs.WorkobjectNo:=0;
            Outputs.PointNo:=0;
            Outputs.UserSpecSpeed1:=0;
            Outputs.UserSpecSpeed2:=0;
            Outputs.Coordinates.X:=0;
            Outputs.Coordinates.Y:=0;
            Outputs.Coordinates.Z:=0;
            Outputs.Coordinates.Rx:=0;
            Outputs.Coordinates.Ry:=0;
            Outputs.Coordinates.Rz:=0;
            Outputs.Start :=FALSE;
            Outputs.Stop:=FALSE;
            Outputs.Pause:=FALSE;
            Outputs.RunAction:=FALSE;
            Outputs.MotorOn:=FALSE;
            _power_progress := 0;
            _movement_progress := 0;
        END_METHOD

        METHOD PUBLIC StartAtMain : IAxoTaskState
            StartAtMain := StartAtMainTask.Invoke(THIS);
        END_METHOD

        METHOD PUBLIC StartMotorsAndProgram : IAxoTaskState
            StartMotorsAndProgram := StartMotorsAndProgramTask.Invoke(THIS);
        END_METHOD

        METHOD PUBLIC StartMovements : IAxoTaskState
            VAR_IN_OUT
                inData : AxoRoboticsMovementsParams;
            END_VAR
            Status.CurrentMovementParameters := inData;

            StartMovements := StartMovementsTask.Invoke(THIS);
        END_METHOD

        METHOD PUBLIC StopMovements : IAxoTaskState
            VAR_INPUT
                inStopType : eAxoRoboticsStopType;
            END_VAR
            _stopType := inStopType;
            StopMovements := StopMovementsTask.Invoke(THIS);
        END_METHOD

        METHOD PUBLIC StopMovementsAndProgram : IAxoTaskState
            VAR_INPUT
                inStopType : eAxoRoboticsStopType;
            END_VAR
            _stopType := inStopType;
            StopMovementsAndProgram := StopMovementsAndProgramTask.Invoke(THIS);
        END_METHOD

        METHOD PRIVATE CallTimers
            VAR_INPUT
                signal : BOOL;
            END_VAR

            _infoTimer.OnDelay(THIS, signal AND Config.InfoTime > LT#0s , Config.InfoTime);
            _errorTimer.OnDelay(THIS, signal AND Config.ErrorTime > LT#0s , Config.ErrorTime );
        END_METHOD

        METHOD PRIVATE GetRobotModeDescription : eAxoUrRoboticsRobotMode
            VAR_INPUT
                inMode:USINT;
            END_VAR
            CASE inMode OF
                USINT#0: GetRobotModeDescription := eAxoUrRoboticsRobotMode#DISCONNECTED;
                USINT#1: GetRobotModeDescription := eAxoUrRoboticsRobotMode#SAFETY;
                USINT#2: GetRobotModeDescription := eAxoUrRoboticsRobotMode#BOOTING;
                USINT#3: GetRobotModeDescription := eAxoUrRoboticsRobotMode#POWER_OFF;
                USINT#4: GetRobotModeDescription := eAxoUrRoboticsRobotMode#POWER_ON;
                USINT#5: GetRobotModeDescription := eAxoUrRoboticsRobotMode#IDLE;
                USINT#6: GetRobotModeDescription := eAxoUrRoboticsRobotMode#BACKDRIVE;
                USINT#7: GetRobotModeDescription := eAxoUrRoboticsRobotMode#RUNNING;
                USINT#8: GetRobotModeDescription := eAxoUrRoboticsRobotMode#UPDATING_FIRMWARE;
            END_CASE;
        END_METHOD
    END_CLASS
END_NAMESPACE
